(* CODESYS project TestSuite_V1.0.8.library
   Author: Simmel Florian
   Version: 1.0.8
   Title: Tc3_PlcTestSuite
   DefaultNamespace: Tc3_PlcTestSuite
   Placeholder: Tc3_PlcTestSuite
   Company: Simmel

Project tree, tasks and I/O mapping:
  libraries: Tc2_Standard, * (Beckhoff Automation GmbH); Tc2_System, * (Beckhoff Automation GmbH); Tc2_Utilities, * (Beckhoff Automation GmbH); Tc3_EventLogger, * (Beckhoff Automation GmbH)
  Interfaces/
    interface I_TestOperation: AssertEqual, ExecuteTest, State, TestId, TestSuiteName
    interface I_TestSuite: ReRunTests, Test
  Project Information/
    function F_GetCompany [ST]
    function F_GetTitle [ST]
    function F_GetVersion [ST]
  Structures/
    data type E_TestStatus
    data type ST_TestDefinition
  Version/
    global variables Global_Version
  function GetValueString [ST]
  global variables GlobalTestSuite
  function block Test [ST]: AssertEqual, ExecuteTest, ReportAssert, State, TestId, TestSuiteName
  function block TestSuite [ST]: ReRunTests, Test, TestSuiteName
  global variables TestSuiteParameter
*)

// Structures/E_TestStatus
{attribute 'qualified_only'}
{attribute 'strict'}
{attribute 'to_string'}
TYPE E_TestStatus : (
		Init := 0,
		Running,
		DoneOk,
		DoneFailed
	);
END_TYPE

// Structures/ST_TestDefinition
TYPE ST_TestDefinition :
	STRUCT
		TestId : T_MaxString;
		Status : E_TestStatus;
	END_STRUCT
END_TYPE

// Version/Global_Version
{attribute 'TcGenerated'}
{attribute 'no-analysis'}
{attribute 'linkalways'}
// This function has been automatically generated from the project information.
VAR_GLOBAL CONSTANT
	{attribute 'const_non_replaced'}
	stLibVersion_Tc3_PlcTestSuite : ST_LibVersion := (iMajor := 1, iMinor := 0, iBuild := 8, iRevision := 0, nFlags := 1, sVersion := '1.0.8');
END_VAR

// GlobalTestSuite
VAR_GLOBAL
	TestSuite : TestSuite<TestSuiteParameter.MaxTestCount>;
END_VAR

// TestSuiteParameter
{attribute 'qualified_only'}
VAR_GLOBAL CONSTANT
	MaxTestCount : DINT := 50;
END_VAR

// Interfaces/I_TestOperation
INTERFACE I_TestOperation EXTENDS __SYSTEM.IQueryInterface

METHOD AssertEqual
VAR_INPUT
	Expected : ANY;
	Actual	 : ANY;
	Epsilon	 : LREAL := 0.000001;
END_VAR
END_METHOD

METHOD ExecuteTest : BOOL
VAR_INPUT
END_VAR
END_METHOD

PROPERTY State : E_TestStatus
GET
END_GET
SET
END_SET
END_PROPERTY

PROPERTY TestId : T_MaxString
GET
END_GET
SET
END_SET
END_PROPERTY

PROPERTY TestSuiteName : String
SET
END_SET
END_PROPERTY

END_INTERFACE

// Interfaces/I_TestSuite
INTERFACE I_TestSuite EXTENDS __SYSTEM.IQueryInterface

METHOD ReRunTests
VAR_INPUT
END_VAR
END_METHOD

METHOD Test : I_TestOperation
VAR_INPUT
	TestId : T_MaxString;
END_VAR
END_METHOD

END_INTERFACE

// Test
FUNCTION_BLOCK Test IMPLEMENTS I_TestOperation
VAR
	_TestSuiteName : STRING;
	_TestId		   : T_MaxString;
	_State		   : E_TestStatus;
	TestMessage	   : FB_TcMessage;
	Source		   : FB_TcSourceInfo;
END_VAR

METHOD AssertEqual
VAR_INPUT
	Expected : ANY;
	Actual	 : ANY;
	Epsilon	 : LREAL := 0.000001;
END_VAR

VAR
	nCount		   : DINT;
	StringExpected : T_MaxString;
	StringActual   : T_MaxString;
	LrealExpected  : LREAL;
	LrealActual	   : LREAL;
	RealExpected   : REAL;
	RealActual	   : REAL;
END_VAR
IF Expected.typeclass <> Actual.typeclass THEN
	State := E_TestStatus.DoneFailed;
	ReportAssert('Type missmatch!');
	RETURN;
END_IF

IF Expected.diSize <> Actual.diSize THEN
	State := E_TestStatus.DoneFailed;
	ReportAssert('Type size missmatch!');
	RETURN;
END_IF

// String
IF Expected.TypeClass = __SYSTEM.TYPE_CLASS.TYPE_ANYSTRING OR Expected.TypeClass = __SYSTEM.TYPE_CLASS.TYPE_STRING OR Expected.TypeClass = __SYSTEM.TYPE_CLASS.TYPE_WSTRING OR Expected.TypeClass = __SYSTEM.TYPE_CLASS.TYPE_XSTRING THEN
	MEMCPY(destAddr := ADR(StringExpected), srcAddr := Expected.pValue, n := DINT_TO_UDINT(Expected.diSize));
	MEMCPY(destAddr := ADR(StringActual), srcAddr := Actual.pValue, n := DINT_TO_UDINT(Actual.diSize));
	IF StringExpected <> StringActual THEN
		State := E_TestStatus.DoneFailed;
		ReportAssert(CONCAT(CONCAT('Expected: ', GetValueString(Expected)), CONCAT(' , Actual: ', GetValueString(Actual))));
		RETURN;
	END_IF
ELSIF Expected.TypeClass = __SYSTEM.TYPE_CLASS.TYPE_LREAL THEN
	MEMCPY(destAddr := ADR(LrealExpected), srcAddr := Expected.pValue, n := DINT_TO_UDINT(Expected.diSize));
	MEMCPY(destAddr := ADR(LrealActual), srcAddr := Actual.pValue, n := DINT_TO_UDINT(Actual.diSize));
	IF ((LrealExpected - Epsilon) > LrealActual) OR ((LrealExpected + Epsilon) < LrealActual) THEN
		State := E_TestStatus.DoneFailed;
		ReportAssert(CONCAT(CONCAT('Expected: ', GetValueString(Expected)), CONCAT(' , Actual: ', GetValueString(Actual))));
		RETURN;
	END_IF
ELSIF Expected.TypeClass = __SYSTEM.TYPE_CLASS.TYPE_ANYREAL OR Expected.TypeClass = __SYSTEM.TYPE_CLASS.TYPE_REAL THEN
	MEMCPY(destAddr := ADR(RealExpected), srcAddr := Expected.pValue, n := DINT_TO_UDINT(Expected.diSize));
	MEMCPY(destAddr := ADR(RealActual), srcAddr := Actual.pValue, n := DINT_TO_UDINT(Actual.diSize));
	IF ((RealExpected - Epsilon) > RealActual) OR ((RealExpected + Epsilon) < RealActual) THEN
		State := E_TestStatus.DoneFailed;
		ReportAssert(CONCAT(CONCAT('Expected: ', GetValueString(Expected)), CONCAT(' , Actual: ', GetValueString(Actual))));
		RETURN;
	END_IF
ELSE
	// Byte comparison
	FOR nCount := 0 TO Actual.diSize - 1 DO
		IF Expected.pvalue[nCount] <> Actual.pvalue[nCount] THEN
			State := E_TestStatus.DoneFailed;
			ReportAssert(CONCAT(CONCAT('Expected: ', GetValueString(Expected)), CONCAT(' , Actual: ', GetValueString(Actual))));
			RETURN;
		END_IF
	END_FOR
END_IF

State := E_TestStatus.DoneOk;
END_METHOD

METHOD ExecuteTest : BOOL
VAR_INPUT
END_VAR
IF State = E_TestStatus.Init THEN
	State := E_TestStatus.Running;
END_IF

ExecuteTest := State = E_TestStatus.Running;
END_METHOD

METHOD PRIVATE ReportAssert
VAR_INPUT
	Reason : STRING := '';
END_VAR

VAR
	ResultString : T_MaxString;
END_VAR
Source.sName := _TestSuiteName;
TestMessage.Create(eventClass	:= TC_EVENT_CLASSES.TestEvents,
				   nEventId		:= 1,
				   eSeverity	:= TcEventSeverity.Error,
				   ipSourceInfo := Source);

ResultString := CONCAT('Test failed - ', TestId);
ResultString := CONCAT(ResultString, '! ');
ResultString := CONCAT(ResultString, Reason);
TestMessage.ipArguments.AddString(ResultString);
TestMessage.Send(0);
Source.Clear();
TestMessage.Release();
END_METHOD

PROPERTY State :  E_TestStatus
GET
State := _State;
END_GET
SET
_State := State;
END_SET
END_PROPERTY

PROPERTY TestId : T_MaxString
GET
TestId := _TestId;
END_GET
SET
_TestId := TestId;
END_SET
END_PROPERTY

PROPERTY TestSuiteName : String
SET
_TestSuiteName := TestSuiteName;
END_SET
END_PROPERTY

END_FUNCTION_BLOCK

// GetValueString
FUNCTION GetValueString : STRING
VAR_INPUT
	Symbol : ANY;
END_VAR

VAR
	ubuff  : ULINT;
	sibuff : SINT;
	ibuff  : INT;
	dibuff : DINT;
	libuff : LINT;
	rbuff  : REAL;
    lrbuff : LREAL;
	sbuff  : STRING(255);
	wsbuff : WSTRING(255);
	x	   : INT; // loop var for STRING and WSTRING
END_VAR

GetValueString := '';
CASE Symbol.TypeClass OF
	__SYSTEM.TYPE_CLASS.TYPE_BOOL:
		memcpy(ADR(ubuff), Symbol.pValue, TO_UDINT(Symbol.diSize));
		GetValueString := TO_STRING(TO_BOOL(TO_LREAL(ubuff)));

	__SYSTEM.TYPE_CLASS.TYPE_BYTE, __SYSTEM.TYPE_CLASS.TYPE_USINT, __SYSTEM.TYPE_CLASS.TYPE_WORD, __SYSTEM.TYPE_CLASS.TYPE_UINT, __SYSTEM.TYPE_CLASS.TYPE_DWORD, __SYSTEM.TYPE_CLASS.TYPE_UDINT, __SYSTEM.TYPE_CLASS.TYPE_LWORD, __SYSTEM.TYPE_CLASS.TYPE_ULINT:
		memcpy(ADR(ubuff), Symbol.pValue, TO_UDINT(Symbol.diSize));
		GetValueString := LREAL_TO_FMTSTR(TO_LREAL(ubuff), 0, FALSE);

	__SYSTEM.TYPE_CLASS.TYPE_SINT:
		memcpy(ADR(sibuff), Symbol.pValue, TO_UDINT(Symbol.diSize));
		GetValueString := LREAL_TO_FMTSTR(TO_LREAL(sibuff), 0, FALSE);

	__SYSTEM.TYPE_CLASS.TYPE_INT:
		memcpy(ADR(ibuff), Symbol.pValue, TO_UDINT(Symbol.diSize));
		GetValueString := LREAL_TO_FMTSTR(TO_LREAL(ibuff), 0, FALSE);

	__SYSTEM.TYPE_CLASS.TYPE_DINT:
		memcpy(ADR(dibuff), Symbol.pValue, TO_UDINT(Symbol.diSize));
		GetValueString := LREAL_TO_FMTSTR(TO_LREAL(dibuff), 0, FALSE);

	__SYSTEM.TYPE_CLASS.TYPE_LINT:
		memcpy(ADR(libuff), Symbol.pValue, TO_UDINT(Symbol.diSize));
		GetValueString := LREAL_TO_FMTSTR(TO_LREAL(libuff), 0, FALSE);

	__SYSTEM.TYPE_CLASS.TYPE_REAL, __SYSTEM.TYPE_CLASS.TYPE_LREAL:
		IF Symbol.TypeClass = __SYSTEM.TYPE_CLASS.TYPE_REAL THEN
			memcpy(ADR(rbuff), Symbol.pValue, TO_UDINT(Symbol.diSize));
			GetValueString := LREAL_TO_FMTSTR(TO_LREAL(rbuff), 5, TRUE);
		ELSIF Symbol.TypeClass = __SYSTEM.TYPE_CLASS.TYPE_LREAL THEN
			memcpy(ADR(lrbuff), Symbol.pValue, TO_UDINT(Symbol.diSize));
			GetValueString := LREAL_TO_FMTSTR(TO_LREAL(lrbuff), 5, TRUE);
		END_IF

	__SYSTEM.TYPE_CLASS.TYPE_STRING, __SYSTEM.TYPE_CLASS.TYPE_WSTRING:
		IF Symbol.TypeClass = __SYSTEM.TYPE_CLASS.TYPE_STRING THEN
			MEMCPY(ADR(sbuff), Symbol.pValue, MIN(SIZEOF(sbuff), TO_UDINT(Symbol.diSize)));
		ELSIF Symbol.TypeClass = __SYSTEM.TYPE_CLASS.TYPE_WSTRING THEN
			MEMCPY(ADR(wsbuff), Symbol.pValue, MIN(SIZEOF(wsbuff), TO_UDINT(Symbol.diSize)));
			WSTRING_TO_STRING2(ADR(sbuff), ADR(wsbuff), SIZEOF(sbuff));
		END_IF

		GetValueString := sbuff;
END_CASE

END_FUNCTION

// Project Information/F_GetCompany
// This function has been automatically generated from the project information.
{attribute 'signature_flag' := '1073741824'}
{attribute 'TcGenerated'}
{attribute 'no-analysis'}
FUNCTION F_GetCompany : WSTRING
VAR_INPUT
	
END_VAR

F_GetCompany := "Simmel";

END_FUNCTION

// Project Information/F_GetTitle
// This function has been automatically generated from the project information.
{attribute 'signature_flag' := '1073741824'}
{attribute 'TcGenerated'}
{attribute 'no-analysis'}
FUNCTION F_GetTitle : WSTRING
VAR_INPUT
	
END_VAR

F_GetTitle := "Tc3_PlcTestSuite";

END_FUNCTION

// Project Information/F_GetVersion
// This function has been automatically generated from the project information.
{attribute 'signature_flag' := '1073741824'}
{attribute 'TcGenerated'}
{attribute 'no-analysis'}
FUNCTION F_GetVersion : ST_LibVersion
VAR_INPUT
	
END_VAR

F_GetVersion.iMajor := 1;
F_GetVersion.iMinor := 0;
F_GetVersion.iBuild := 8;
F_GetVersion.iRevision := 0;
F_GetVersion.sVersion := '1.0.8';
F_GetVersion.nFlags := 1;

END_FUNCTION

// TestSuite
FUNCTION_BLOCK TestSuite 
VAR_GENERIC CONSTANT
    _MaxTestCount : DINT := 10;
END_VAR
IMPLEMENTS I_TestSuite
VAR
    _TestSuiteName    : STRING;
	TestCollection	  : ARRAY[0.._MaxTestCount] OF Test;
	NoAction		  : Test := (TestId := 'No Action', State := E_TestStatus.DoneOk);
	ActiveTest		  : DINT;
	DoneMessage		  : FB_TcMessage;
    Source            : FB_TcSourceInfo;
	TotalTestCount	  : UDINT := 0;
	TotalOkTestCount  : UDINT := 0;
	TotalNokTestCount : UDINT := 0;
	Complete		  : BOOL;
END_VAR

METHOD ReRunTests
VAR
	i : DINT;
END_VAR
FOR i := 0 TO TestSuiteParameter.MaxTestCount DO
	TestCollection[i].State := E_TestStatus.Init;
	ActiveTest				:= 0;
	Complete				:= FALSE;
END_FOR
END_METHOD

METHOD Test : I_TestOperation
VAR_INPUT
	TestId : T_MaxString;
END_VAR

VAR
	ResultString : T_MaxString;
	i			 : DINT;
END_VAR
IF _TestSuiteName = '' THEN
	_TestSuiteName := __POUNAME();
END_IF

IF NOT Complete THEN
	FOR i := 0 TO _MaxTestCount DO
		TestCollection[i].TestSuiteName := _TestSuiteName;

		// Detect first running test
		IF TestCollection[i].State = E_TestStatus.Running THEN
			ActiveTest := i;
		END_IF

		IF TestCollection[ActiveTest].State >= E_TestStatus.DoneOk THEN
			ActiveTest := 0;
		END_IF

		// Get existing Test
		IF (TestCollection[i].TestId = TestId) THEN
			IF (ActiveTest = i) OR (ActiveTest = 0) THEN
				Test := TestCollection[i];
			ELSE
				Test := NoAction;
			END_IF

			EXIT;
		END_IF

		// Add Test
		IF TestCollection[i].TestId = '' THEN
			TestCollection[i].TestId := TestId;
			Test					 := NoAction;
			EXIT;
		END_IF

		// Out of tests
		IF i = _MaxTestCount THEN
			Test		 := NoAction;
			Source.sName := _TestSuiteName;
			DoneMessage.Create(eventClass	:= TC_EVENT_CLASSES.TestEvents,
							   nEventId		:= 1,
							   eSeverity	:= TcEventSeverity.Error,
							   ipSourceInfo := Source);

			ResultString := CONCAT('Test not added, max Tests exeeded - ', TO_STRING(_MaxTestCount));
			DoneMessage.ipArguments.AddString(ResultString);
			DoneMessage.Send(0);
			Source.Clear();
			DoneMessage.Release();
			Complete := TRUE;
		END_IF
	END_FOR

	// Run Statistic
	TotalTestCount	  := 0;
	TotalOkTestCount  := 0;
	TotalNokTestCount := 0;
	FOR i := 0 TO _MaxTestCount DO
		IF TestCollection[i].TestId <> '' THEN
			TotalTestCount := TotalTestCount + 1;
			IF TestCollection[i].State = E_TestStatus.DoneOk THEN
				TotalOkTestCount := TotalOkTestCount + 1;
			END_IF

			IF TestCollection[i].State = E_TestStatus.DoneFailed THEN
				TotalNokTestCount := TotalNokTestCount + 1;
			END_IF
		END_IF
	END_FOR

	// Tests finished
	IF (TotalTestCount = (TotalOkTestCount + TotalNokTestCount)) AND NOT Complete THEN
		Source.sName := _TestSuiteName;
		DoneMessage.Create(eventClass	:= TC_EVENT_CLASSES.TestEvents,
						   nEventId		:= 1,
						   eSeverity	:= TcEventSeverity.Error,
						   ipSourceInfo := Source);

		ResultString := CONCAT('Completed - ', CONCAT('Total Tests - ', TO_STRING(TotalTestCount)));
		ResultString := CONCAT(ResultString, CONCAT(', OK Tests - ', TO_STRING(TotalOkTestCount)));
		ResultString := CONCAT(ResultString, CONCAT(', Failed Tests - ', TO_STRING(TotalNokTestCount)));
		DoneMessage.ipArguments.AddString(ResultString);
		DoneMessage.Send(0);
		Source.Clear();
		DoneMessage.Release();
		Complete := TRUE;
	END_IF
ELSE
	Test := NoAction;
END_IF
END_METHOD

PROPERTY TestSuiteName : String
SET
_TestSuiteName := TestSuiteName;
END_SET
END_PROPERTY

END_FUNCTION_BLOCK
